// TIA Portal V19 export
VAR_GLOBAL   // PLC tag table "tags_IO"
   "866TR2510-S1_Rev" AT %I0.0 : Bool;   // 866TR2510 - Reverse KP-208
   "866TR2510-S1_Fwd" AT %I0.1 : Bool;   // 866TR2510 - Forward KP-208
   "866TR2520-S1_Rev" AT %I0.2 : Bool;   // 866TR2520 - Reverse KP-208
   "866TR2520-S1_Fwd" AT %I0.3 : Bool;   // 866TR2520 - Forward KP-208
   "866TR2530-S1_Rev" AT %I0.4 : Bool;   // 866TR2530 - Reverse KP-208
   "866TR2530-S1_Fwd" AT %I0.5 : Bool;   // 866TR2530 - Forward KP-208
   "866LE2540-S1_Up" AT %I0.6 : Bool;   // 866LE2540 - Cage up
   "866LE2540-S1_Down" AT %I0.7 : Bool;   // 866LE2540 - Cage down
   "866TR2541-S1_Rev" AT %I1.0 : Bool;   // 866TR2541 - Reverse KP-208
   "866TR2541-S1_Fwd" AT %I1.1 : Bool;   // 866TR2541 - Forward KP-208
   "866TR2542-S1_Rev" AT %I1.2 : Bool;   // 866TR2542 - Reverse
   "866TR2542-S1_Fwd" AT %I1.3 : Bool;   // 866TR2542 - Forward
   "866MA2543-S1_In" AT %I1.4 : Bool;   // 866MA2543 - In
   "866MA2543-S1_Out" AT %I1.5 : Bool;   // 866MA2543 - Out
   "866TR2510-GL1" AT %I1.6 : Bool;   // 866TR2510 - Entry photocell
   "866TR2510-GL2" AT %I1.7 : Bool;   // 866TR2510 - Exit photocell
   "866TR2520-GL1" AT %I2.0 : Bool;   // 866TR2520 - Entry photocell
   "866TR2520-GL2" AT %I2.1 : Bool;   // 866TR2520 - Exit photocell
   "866TR2530-GL1" AT %I2.2 : Bool;   // 866TR2530 - Entry photocell
   "866TR2530-GL2" AT %I2.3 : Bool;   // 866TR2530 - Exit photocell
   "2510_KontrollOrd" AT %QW400 : Word;
   "2510_StatusOrd" AT %IW400 : Word;
   "2510_SpeedSP" AT %QW402 : Word;
   "2510_SpeedPV" AT %IW402 : Word;
   "2520_KontrollOrd" AT %QW388 : Word;
   "2520_StatusOrd" AT %IW388 : Word;
   "2520_SpeedSP" AT %QW390 : Word;
   "2520_SpeedPV" AT %IW390 : Word;
   "2530_KontrollOrd" AT %QW376 : Word;
   "2530_StatusOrd" AT %IW376 : Word;
   "2530_SpeedSP" AT %QW378 : Word;
   "2530_SpeedPV" AT %IW378 : Word;
   "2600_KontrollOrd" AT %QW412 : Word;
   "2600_StatusOrd" AT %IW412 : Word;
   "2600_SpeedSP" AT %QW414 : Word;
   "2600_SpeedPV" AT %IW414 : Word;
   "101LT1" AT %IW100 : Word;   // Tank 101 Level transmitter 1
   "101LT2" AT %IW102 : Word;   // Tank 101 Level transmitter 2
   "102LT1" AT %IW104 : Word;   // Tank 102 Level transmitter 1
   "102LT2" AT %IW106 : Word;   // Tank 102 Level transmitter 2
   "101CV1" AT %QW100 : Word;   // Tank 101 Control valve 1
   "101CV2" AT %QW102 : Word;   // Tank 101 Control valve 2
   "102CV1" AT %QW104 : Word;   // Tank 102 Control valve 1
   "102CV2" AT %QW106 : Word;   // Tank 102 Control valve 2
   "101PT1" AT %IW108 : Word;   // Tank 101 Pressure transmitter 1
   "101PT2" AT %IW110 : Word;   // Tank 101 Pressure transmitter 2
   "102PT1" AT %IW112 : Word;   // Tank 102 Pressure transmitter 1
   "102PT2" AT %IW114 : Word;   // Tank 102 Pressure transmitter 2
   "101FT1" AT %IW116 : Word;   // Tank 101 Flow transmitter 1
   "101FT2" AT %IW118 : Word;   // Tank 101 Flow transmitter 2
   "102FT1" AT %IW120 : Word;   // Tank 102 Flow transmitter 1
   "102FT2" AT %IW122 : Word;   // Tank 102 Flow transmitter 2
   "101DV1_GL1" AT %I3.0 : Bool;   // 101DV1 Digital valve open feedback
   "101DV1_GL2" AT %I3.1 : Bool;   // 101DV1 Digital valve closed feedback
   "101DV2_GL1" AT %I3.2 : Bool;   // 101DV2 Digital valve open feedback
   "101DV2_GL2" AT %I3.3 : Bool;   // 101DV2 Digital valve closed feedback
   "101DV1_OPEN" AT %Q0.0 : Bool;
   "101DV2_OPEN" AT %Q0.1 : Bool;
END_VAR
